FUNCTION F_ClearLarge 
VAR_IN_OUT CONSTANT
	stringToClear 	: STRING(StringsParams.MAX_STRING_LENGTH);
END_VAR

MEMSET(ADR(stringToClear), 16#0, sizeof(stringToClear));

END_FUNCTION

(* stored: Version 1.1.0.1, ProductVersion 3.1.4022.6
   POU F_ClearLarge: Id {aee1f00c-288c-495e-9191-3d47b22ee060}, SpecialFunc None *)
